// TIA Portal V18 export
DATA_BLOCK "Data_block_1"   // DB26
{ S7_Optimized_Access := 'TRUE' }
VERSION : 0.1
// stored: AutoNumber true, DBAccessibleFromOPCUA true, IsOnlyStoredInLoadMemory false, IsRetainMemResEnabled false, IsWriteProtectedInAS false, MemoryReserve 100
   VAR
      on : Bool;
      outmin : Int;
      outhout : Int;
   END_VAR
BEGIN
END_DATA_BLOCK
